// TwinCAT 3 PLC project Sandbox
// ProgramVersion: 3.1.4024.12
// libraries:
//   Tc2_Standard, * (Beckhoff Automation GmbH)
//   Tc2_System, * (Beckhoff Automation GmbH)
//   Tc3_Module, * (Beckhoff Automation GmbH)
//   TcUnit, * (www.tcunit.org)
// project tree:
//   Functional FBs/ BrokenCalculator.TcPOU, Calculator.TcPOU
//   Interfaces/ ISum.TcIO, ISumTest.TcIO
//   / PlcTask.TcTTO
//   Main/ MAIN.TcPOU
//   TestSuites/ BrokenCalculatorTest.TcPOU, CalculatorTest.TcPOU, SumTest.TcPOU, TestSuite.TcPOU
// real-time tasks:
//   TASK PlcTask: cycle T#10ms, priority 20, ADS port 350

CONFIGURATION Sandbox
    RESOURCE PLC ON TwinCAT3
        TASK PlcTask(INTERVAL := T#10ms, PRIORITY := 20);
        PROGRAM MAIN WITH PlcTask : MAIN;
    END_RESOURCE
END_CONFIGURATION

// ---- Interfaces/ISum.TcIO
INTERFACE ISum

(*This method adds two DINT numbers and returns the result in Sum*)
METHOD Sum : DINT;
VAR_INPUT
	Dint1 : DINT;
	Dint2 : DINT;
END_VAR
END_METHOD

END_INTERFACE

// ---- Interfaces/ISumTest.TcIO
INTERFACE ISumTest

(*This method is used to prepare arrays with dint1 dint2 and expected dints*)
METHOD prepareSumTest : BOOL
VAR_INPUT
END_VAR
END_METHOD

END_INTERFACE

// ---- Main/MAIN.TcPOU
PROGRAM MAIN
VAR
	TestSuite : TestSuite;
	CalculatorTest : CalculatorTest;
	BrokenCalculatorTest: BrokenCalculatorTest;
END_VAR

TcUnit.RUN();

END_PROGRAM

// ---- TestSuites/TestSuite.TcPOU
FUNCTION_BLOCK TestSuite EXTENDS FB_TestSuite

END_FUNCTION_BLOCK

// ---- TestSuites/CalculatorTest.TcPOU
FUNCTION_BLOCK CalculatorTest EXTENDS FB_TestSuite IMPLEMENTS ISumTest
VAR
	_dint1s : ARRAY[0..2] OF DINT;
	_dint2s : ARRAY[0..2] OF DINT;
	_expected : ARRAY[0..2] OF DINT;
	_adders : ARRAY[0..2] OF ISum;
	sumtest : SumTest;
END_VAR

prepareSumTest();
sumtest(Dint1s := _dint1s, Dint2s := _dint2s, expected := _expected, adders := _adders);

{warning 'add method implementation '}
(*This method is used to prepare arrays with dint1 dint2 and expected dints*)
METHOD prepareSumTest : BOOL
VAR_INST
	adder0 : Calculator;
	adder1 : Calculator;
	adder2 : Calculator;
END_VAR
_dint1s[0] := 0;
_dint2s[0] := 5;
_expected[0] := 5;
_adders[0] := adder0;

_dint1s[1] := 5;
_dint2s[1] := 0;
_expected[1] := 5;
_adders[1] := adder1;

_dint1s[2] := 45;
_dint2s[2] := 2;
_expected[2] := 47;
_adders[2] := adder2;
END_METHOD

END_FUNCTION_BLOCK

// ---- TestSuites/SumTest.TcPOU
FUNCTION_BLOCK SumTest EXTENDS FB_TestSuite
VAR_INPUT
	Dint1s : ARRAY[0..2] OF DINT;
	Dint2s : ARRAY[0..2] OF DINT;
	expected : ARRAY[0..2] OF DINT;
	adders : ARRAY[0..2] OF ISum;
END_VAR

addingTest('test0', Dint1s[0], Dint2s[0], expected[0], adders[0]);
addingTest('test1', Dint1s[1], Dint2s[1], expected[1], adders[1]);
addingTest('test2', Dint1s[2], Dint2s[2], expected[2], adders[2]);

METHOD addingTest
VAR_INPUT
	testName : STRING;
	dint1 : DINT;
	dint2 : DINT;
	expected : DINT;
	adder : ISum;
END_VAR
VAR
	actual : DINT;
END_VAR
TEST(testName);

actual := adder.Sum(dint1, dint2);
AssertEquals(expected, actual, 'The result was not like expected');
TEST_FINISHED();
END_METHOD

END_FUNCTION_BLOCK

// ---- Functional FBs/Calculator.TcPOU
FUNCTION_BLOCK Calculator IMPLEMENTS ISum

METHOD Sum : DINT
VAR_INPUT
	Dint1 : DINT;
	Dint2 : DINT;
END_VAR
Sum := Dint1 + Dint2;
END_METHOD

END_FUNCTION_BLOCK

// ---- TestSuites/BrokenCalculatorTest.TcPOU
FUNCTION_BLOCK BrokenCalculatorTest EXTENDS FB_TestSuite IMPLEMENTS ISumTest
VAR
	_dint1s : ARRAY[0..2] OF DINT;
	_dint2s : ARRAY[0..2] OF DINT;
	_expected : ARRAY[0..2] OF DINT;
	_adders : ARRAY[0..2] OF ISum;
	sumtest : SumTest;
END_VAR

prepareSumTest();
sumtest(Dint1s := _dint1s, Dint2s := _dint2s, expected := _expected, adders := _adders);

{warning 'add method implementation '}
(*This method is used to prepare arrays with dint1 dint2 and expected dints*)
METHOD prepareSumTest : BOOL
VAR_INST
	adder0 : BrokenCalculator;
	adder1 : BrokenCalculator;
	adder2 : BrokenCalculator;
END_VAR
_dint1s[0] := 0;
_dint2s[0] := 5;
_expected[0] := 5;
_adders[0] := adder0;

_dint1s[1] := 5;
_dint2s[1] := 0;
_expected[1] := 5;
_adders[1] := adder1;

_dint1s[2] := 45;
_dint2s[2] := 2;
_expected[2] := 47;
_adders[2] := adder2;
END_METHOD

END_FUNCTION_BLOCK

// ---- Functional FBs/BrokenCalculator.TcPOU
FUNCTION_BLOCK BrokenCalculator IMPLEMENTS ISum

(*This method adds two DINT numbers and returns the result in Sum*)
METHOD Sum : DINT
VAR_INPUT
	Dint1 : DINT;
	Dint2 : DINT;
END_VAR
Sum := Dint1 * Dint2;
END_METHOD

END_FUNCTION_BLOCK
